Fanuc KAREL source: CA0015.KL

PROGRAM CA0015
%STACKSIZE=65535
%PRIORITY=65535
%NOLOCKGROUP
TYPE
T=STRUCTURE
A : INTEGER
B : REAL
ENDSTRUCTURE
VAR
G : INTEGER
I : INTEGER
R : REAL
B : BOOLEAN
S : STRING[16]
AI : ARRAY[2] OF INTEGER
AR : ARRAY[2] OF REAL
ST : T
P : XYZWPR
V : VECTOR
ROUTINE F(P1 : INTEGER; P2 : REAL; P3 : BOOLEAN) FROM CA0015
ROUTINE F
BEGIN
G=(G + 1)
END F
BEGIN
G=0
I=1
R=2.5
B=TRUE
S='A'
AI[1]=3
AR[1]=4.5
-- UNSAFE_SOURCE_IR line 33: ST.A = 5
-- UNSAFE_SOURCE_IR line 34: ST.B = 6.5
F(I,R,B)
END CA0015
